(* function to calculate trigger points for time based moves *)
FUNCTION F_TriggerPosOffset : LREAL
VAR_INPUT
	Velocity		: LREAL	; // [Units/sec] command velocity 
	nMoveTimeMs		: LREAL	; // [ms] Time it takes for move to complete
END_VAR
VAR
END_VAR

// ===== Convert time to usable calculation value =====
	F_TriggerPosOffset := nMovetimeMs * ABS(Velocity / 1000);

END_FUNCTION

(* stored: Version 1.1.0.1, ProductVersion 3.1.4024.3
   POU F_TriggerPosOffset: Id {b2f198b1-9b50-4852-9d0f-5e1a8aa42ff7}, SpecialFunc None *)
